// TIA Portal V20 export
DATA_BLOCK "DB_AsiSetpoint"   // DB24
// stored: Access Published, MemoryReserve 100, Namespace LineB1
   VAR
      Line : Struct
         B1 : Struct
            DirChange : Struct
               Conveyor : Array[_.minB1.._.maxB1] of Bool;
            END_STRUCT;
            Speed : Struct
               Conveyor : Array[_.minB1.._.maxB1] of Bool;
            END_STRUCT;
         END_STRUCT;
      END_STRUCT;
   END_VAR
BEGIN
END_DATA_BLOCK
